FUNCTION IsValueEven : BOOL
VAR_INPUT
	Value : ANY_INT;
END_VAR
VAR
	pAnyUSINT : POINTER TO USINT; 
	pAnyUINT : POINTER TO UINT;
	pAnyUDINT : POINTER TO UDINT; 
	pAnyULINT : POINTER TO ULINT;
	pAnySINT : POINTER TO SINT; 
	pAnyINT : POINTER TO INT;
	pAnyDINT : POINTER TO DINT; 
	pAnyLINT : POINTER TO LINT;
	conversion : ULINT;
END_VAR

IF (Value.TypeClass = __SYSTEM.TYPE_CLASS.TYPE_USINT) THEN
    pAnyUSINT := Value.pValue; 
    conversion  := USINT_TO_ULINT(pAnyUSINT^);
	
ELSIF (Value.TypeClass = __SYSTEM.TYPE_CLASS.TYPE_UINT) THEN
    pAnyUINT := Value.pValue; 
    conversion  := UINT_TO_ULINT(pAnyUINT^);
	
ELSIF (Value.TypeClass = __SYSTEM.TYPE_CLASS.TYPE_UDINT) THEN
    pAnyUDINT := Value.pValue; 
    conversion  := UDINT_TO_ULINT(pAnyUDINT^);
	
ELSIF (Value.TypeClass = __SYSTEM.TYPE_CLASS.TYPE_ULINT) THEN
    pAnyULint := Value.pValue; 
    conversion  := pAnyULint^;
	
ELSIF (Value.TypeClass = __SYSTEM.TYPE_CLASS.TYPE_SINT) THEN
    pAnySINT := Value.pValue; 
    conversion  := SINT_TO_ULINT(pAnySINT^);
	
ELSIF (Value.TypeClass = __SYSTEM.TYPE_CLASS.TYPE_INT) THEN
    pAnyINT := Value.pValue; 
    conversion  := INT_TO_ULINT(pAnyINT^);
	
ELSIF (Value.TypeClass = __SYSTEM.TYPE_CLASS.TYPE_DINT) THEN
    pAnyDINT := Value.pValue; 
    conversion  := DINT_TO_ULINT(pAnyDINT^);
	
ELSIF (Value.TypeClass = __SYSTEM.TYPE_CLASS.TYPE_LINT) THEN
    pAnyLINT := Value.pValue; 
    conversion  := LINT_TO_ULINT(pAnyLINT^);

ELSE
	RETURN;
	
END_IF;

IsValueEven := (conversion MOD 2 ) = 0;

END_FUNCTION

(* stored: Version 1.1.0.1, ProductVersion 3.1.4024.12
   POU IsValueEven: Id {8600193d-18ce-0c34-227e-45c7aedf4949}, SpecialFunc None *)
